FUNCTION BYTES_TO_ARR08B (* this Function combines 8 BYTEs to a 8-BYTE Array *)
  (* Standard: 61499-1; Description: Copyright (c) 2024 HR Agrartechnik GmbH This program and the accompanying materials are made available under the terms of the Eclipse Public License 2.0 which is available at https://www.eclipse.org/legal/epl-2.0/ SPDX-License-Identifier: EPL-2.0 *)
  (* Version 1.0, 2024-02-22, Franz Höpfinger, HR Agrartechnik GmbH *)
  PACKAGE logiBUS::utils::conversion::arr::reversing;
  IMPORT eclipse4diac::core::TypeHash;
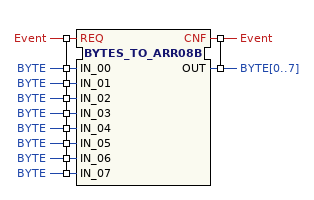
  EVENT_INPUT
    REQ WITH IN_00, IN_01, IN_02, IN_03, IN_04, IN_05, IN_06, IN_07;
  END_EVENT
  EVENT_OUTPUT
    CNF WITH OUT;
  END_EVENT
  VAR_INPUT
    IN_00 : BYTE; (* BYTE 00 *)
    IN_01 : BYTE; (* BYTE 01 *)
    IN_02 : BYTE; (* BYTE 02 *)
    IN_03 : BYTE; (* BYTE 03 *)
    IN_04 : BYTE; (* BYTE 04 *)
    IN_05 : BYTE; (* BYTE 05 *)
    IN_06 : BYTE; (* BYTE 06 *)
    IN_07 : BYTE; (* BYTE 07 *)
  END_VAR
  VAR_OUTPUT
    OUT : ARRAY [0..7] OF BYTE; (* ARR08B Output *)
  END_VAR
  BODY IN ST:
PACKAGE logiBUS::utils::conversion::arr::reversing;

(* this Function combines 8 BYTEs to a 8-BYTE Array *)
FUNCTION BYTES_TO_ARR08B

VAR_INPUT
	IN_00 : BYTE; // BYTE 00
	IN_01 : BYTE; // BYTE 01
	IN_02 : BYTE; // BYTE 02
	IN_03 : BYTE; // BYTE 03
	IN_04 : BYTE; // BYTE 04
	IN_05 : BYTE; // BYTE 05
	IN_06 : BYTE; // BYTE 06
	IN_07 : BYTE; // BYTE 07
END_VAR

VAR_OUTPUT
	OUT : ARRAY[0..7] OF BYTE; // ARR08B Output
END_VAR

OUT[0] := IN_00;
OUT[1] := IN_01;
OUT[2] := IN_02;
OUT[3] := IN_03;
OUT[4] := IN_04;
OUT[5] := IN_05;
OUT[6] := IN_06;
OUT[7] := IN_07;

END_FUNCTION
  END_BODY
END_FUNCTION
